FUNCTION_BLOCK FB_Cargar_SFC

VAR_INPUT
    // SFC-Flags
    SFCPause: BOOL;
    SFCReset: BOOL;
     
    // Sincronizacion
    Benido: BOOL ;
    Ejecuta: BOOL;
    
    CargadorDetras AT %I* : BOOL;
    CargadorDelante AT %I* : BOOL;
    CargadorArriba AT %I* : BOOL;
    CargadorAbajo AT %I* : BOOL;
END_VAR
VAR_OUTPUT
     // Sincronizacion    
    Acabhe: BOOL;
    ListoKalisto: BOOL;
    
  	//CargadorAvanza AT %Q* : BOOL;
    //CargadorBaja AT %Q* : BOOL;
  //  CargadorCierra AT %Q* : BOOL;
    
    CargadorAvanza: BOOL;
    CargadorBaja: BOOL;
    CargadorCierra: BOOL;
END_VAR

VAR_IN_OUT
  Tapas : ARRAY[0..7] OF ST_POSICION;
END_VAR

VAR 
END_VAR

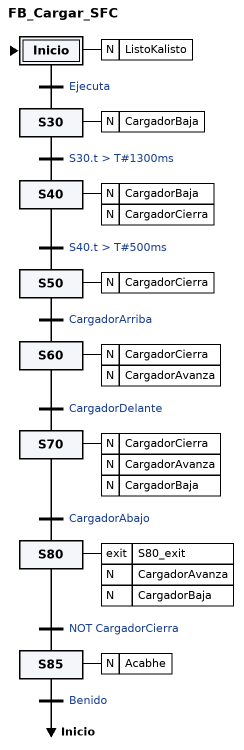
INITIAL_STEP Inicio:
    ListoKalisto(N);
END_STEP
TRANSITION FROM Inicio TO S30
    := Ejecuta;
END_TRANSITION
STEP S30:
    CargadorBaja(N);
END_STEP
TRANSITION FROM S30 TO S40
    := S30.t > T#1300ms;
END_TRANSITION
STEP S40:
    CargadorBaja(N);
    CargadorCierra(N);
END_STEP
TRANSITION FROM S40 TO S50
    := S40.t > T#500ms;
END_TRANSITION
STEP S50:
    CargadorCierra(N);
END_STEP
TRANSITION FROM S50 TO S60
    := CargadorArriba;
END_TRANSITION
STEP S60:
    CargadorCierra(N);
    CargadorAvanza(N);
END_STEP
TRANSITION FROM S60 TO S70
    := CargadorDelante;
END_TRANSITION
STEP S70:
    CargadorCierra(N);
    CargadorAvanza(N);
    CargadorBaja(N);
END_STEP
TRANSITION FROM S70 TO S80
    := CargadorAbajo;
END_TRANSITION
STEP S80:
    S80_exit(P0);  // exit action
    CargadorAvanza(N);
    CargadorBaja(N);
END_STEP
TRANSITION FROM S80 TO S85
    := NOT CargadorCierra;
END_TRANSITION
STEP S85:
    Acabhe(N);
END_STEP
TRANSITION FROM S85 TO Inicio
    := Benido;
END_TRANSITION

ACTION S80_exit:
Tapas[0].Ocupada := TRUE;
END_ACTION

END_FUNCTION_BLOCK

(* stored: Version 1.1.0.1, ProductVersion 3.1.4024.12
   POU FB_Cargar_SFC: Id {7e010383-13df-4e7d-9795-68d3bb4c108c}, SpecialFunc None
   Action S80_exit: Id {7fd38af6-6564-488d-b9c0-8d1282b38353} *)
